(* PLC project Modbus, Beremiz Beremiz 1 *)
(* stored: creationDateTime 2018-07-27T13:19:12, modificationDateTime 2018-07-27T15:43:56 *)

FUNCTION_BLOCK Generator
  VAR_OUTPUT
    OUT : BOOL;
  END_VAR
  VAR_INPUT
    PON : TIME;
    POFF : TIME;
  END_VAR
  VAR
    T1 : TON;
    T2 : TOF;
  END_VAR

            T1( IN := NOT T2.Q, PT := POFF);
T2( IN := T1.Q,     PT := PON);
OUT := T2.Q;
          
END_FUNCTION_BLOCK

PROGRAM program0
  VAR
    Counter : INT;
    CounterReadBack : INT;
  END_VAR
  VAR
    MasterWriteToReg0 AT %QW0.0.0.0 : INT;
    MasterReadFromReg1 AT %IW0.0.1.0 : INT;
    SlaveHoldReg0 AT %IW0.1.0.0 : WORD;
    SlaveInputReg0 AT %QW0.1.1.0 : WORD;
  END_VAR
  VAR
    CTU0 : CTU;
    Generator0 : Generator;
  END_VAR
  VAR  (* added by the conversion: wires and edge detectors of the diagram *)
    R_TRIG1 : R_TRIG;
  END_VAR

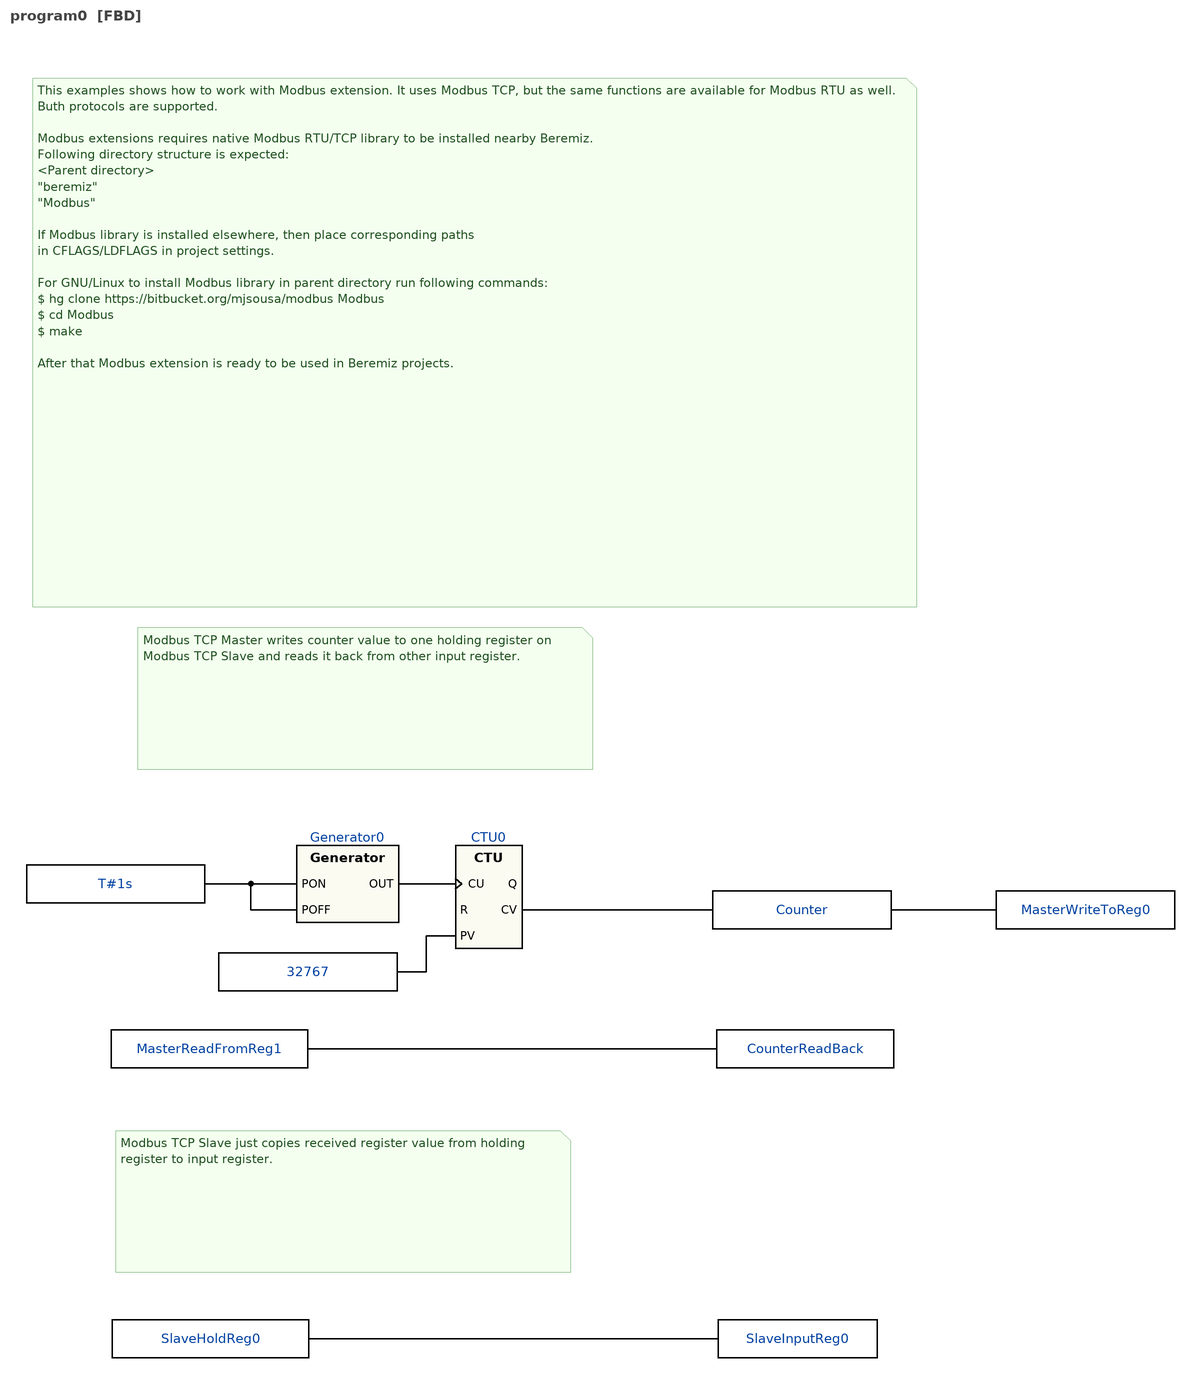
(* FBD diagram, written out as Structured Text *)
(* This examples shows how to work with Modbus extension. It uses Modbus TCP, but the same functions are available for Modbus RTU as well. Buth protocols are supported.

Modbus extensions requires native Modbus RTU/TCP library to be installed nearby Beremiz.
Following directory structure is expected:
<Parent directory>
  "beremiz"
  "Modbus"

If Modbus library is installed elsewhere, then place corresponding paths
in CFLAGS/LDFLAGS in project settings.

For GNU/Linux to install Modbus library in parent directory run following commands:
$ hg clone https://bitbucket.org/mjsousa/modbus Modbus
$ cd Modbus
$ make

After that Modbus extension is ready to be used in Beremiz projects. *)
(* Modbus TCP Master writes counter value to one holding register on Modbus TCP Slave and reads it back from other input register. *)
Generator0(PON := T#1s, POFF := T#1s);
R_TRIG1(CLK := Generator0.OUT);
CTU0(CU := R_TRIG1.Q, PV := 32767);
Counter := CTU0.CV;
MasterWriteToReg0 := Counter;
CounterReadBack := MasterReadFromReg1;
(* Modbus TCP Slave just copies received register value from holding register to input register. *)
SlaveInputReg0 := SlaveHoldReg0;
END_PROGRAM

CONFIGURATION config
  RESOURCE resource1 ON PLC
    TASK task0(INTERVAL := T#20ms, PRIORITY := 0);
    PROGRAM instance0 WITH task0 : program0;
  END_RESOURCE
END_CONFIGURATION
